FUNCTION_BLOCK DFB_Second_Pulse
VAR_INPUT
	TON1_TIME: TIME;
END_VAR
VAR_OUTPUT
	QSec_P: BOOL;
END_VAR
VAR
	fb_TON1: TON;
END_VAR

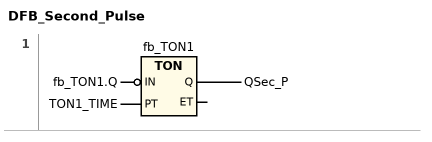
// NETWORK 1
fb_TON1(IN := NOT fb_TON1.Q, PT := TON1_TIME); // TON
QSec_P := fb_TON1.Q;

END_FUNCTION_BLOCK

(* stored: Version 1.1.0.1, ProductVersion 3.1.4022.18
   POU DFB_Second_Pulse: Id {be561450-d5f5-4644-bda8-4743a3d521ce}, SpecialFunc None *)
